RoboDK station: Group9-Robotics.rdk

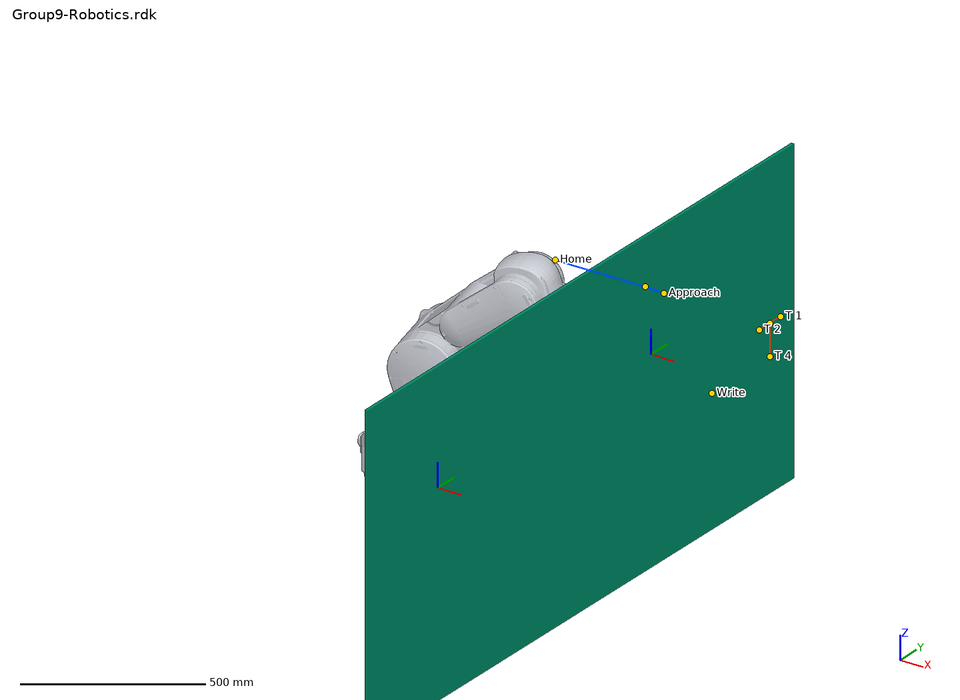
[picture v0: the station drawn from its stored meshes, robots at their saved joint values, targets as dots, program paths as lines]
Station ProjectWrite5 (saved by RoboDK 5.6.8). Poses are relative to the parent item; angles as X-Y-Z fixed-axis rotations.
Station parameters (name, value as stored): red, -1
  - frame Mitsubishi RV-7FR Base at (0, 0, 0) mm
    - robot Mitsubishi RV-7FR: 6 axes, payload 7 kg, reach 713 mm, repeatability 0.02 mm, weight 65 kg
        modified DH rows (alpha deg, a mm, theta deg, d mm): 0, 0, 0, 400; -90, 0, -90, 0; 0, 340, -90, 0; -90, 50, 0, 370; 90, 0, 0, 0; -90, 0, 180, 85
        joint limits [-240, -115, 0, -200, -120, -360] to [240, 125, 156, 200, 120, 360]; home [0, 0, 90, 0, 0, 0]; saved at [13.788, 47.313, 119.158, 14.166, -76.867, 176.718]
      - tool Tool, TCP at (0, 0, 283) mm, rotated rx 0 ry 0 rz -90 deg, size 100 x 89.2 x 281.5 mm
  - frame Frame 2 at (0, 1000, 0) mm
    - target Approach (Cartesian target) at (742, -1000, 790) mm, rotated rx 90 ry 0 rz 90 deg; joints [0, 0.675, 89.322, 180, -0.004, 0] of Mitsubishi RV-7FR
    - target Home (Cartesian target) at (386.81, -1000, 790) mm, rotated rx 90 ry 0 rz 90 deg; joints [0, -58.255, 121.519, 180, -26.736, 0] of Mitsubishi RV-7FR
    - target Write (Cartesian target) at (742, -775, 400) mm, rotated rx 90 ry 0 rz 90 deg; joints [31.031, 34.171, 112.413, 35.782, -61.843, 161.216] of Mitsubishi RV-7FR
    - target Retract (Cartesian target) at (680.67, -1000, 792.94) mm, rotated rx 90 ry 0 rz 90 deg; joints [0, -9.518, 98.336, 180, -1.182, 0] of Mitsubishi RV-7FR
    - target T 1 (Cartesian target) at (740, -450, 500) mm, rotated rx 0 ry 90 rz 0 deg; joints [55.927, 60.719, 47.204, 78.242, -57.788, -68.671] of Mitsubishi RV-7FR
    - target T 2 (Cartesian target) at (740, -550, 500) mm, rotated rx 0 ry 90 rz 0 deg; joints [50.421, 44.575, 75.507, 67.493, -56.542, -53.073] of Mitsubishi RV-7FR
    - target T 3 (Cartesian target) at (740, -500, 500) mm, rotated rx 0 ry 90 rz 0 deg; joints [53.351, 51.664, 63.311, 72.561, -57.241, -59.863] of Mitsubishi RV-7FR
    - target T 4 (Cartesian target) at (740, -500, 400) mm, rotated rx 0 ry 90 rz 0 deg; joints [53.351, 59.352, 66.003, 66.708, -60.867, -48.513] of Mitsubishi RV-7FR
  - object Board2mX1m at (740, -400, 1000) mm, rotated rx -90 ry 0 rz -90 deg, size 2000 x 1000 x 10 mm, geometry from Board2mX1m.STEP
  - program Prog1 (8 instructions, listed below)
  - Python program WriteRobodk (listed below)
  - program Prog3 (7 instructions, listed below)
  - Python program TimesNewRoman (listed below)
  - program Main Prog (3 instructions, listed below)
  - Python program WeldOff (listed below)
  - Python program WeldOn (listed below)
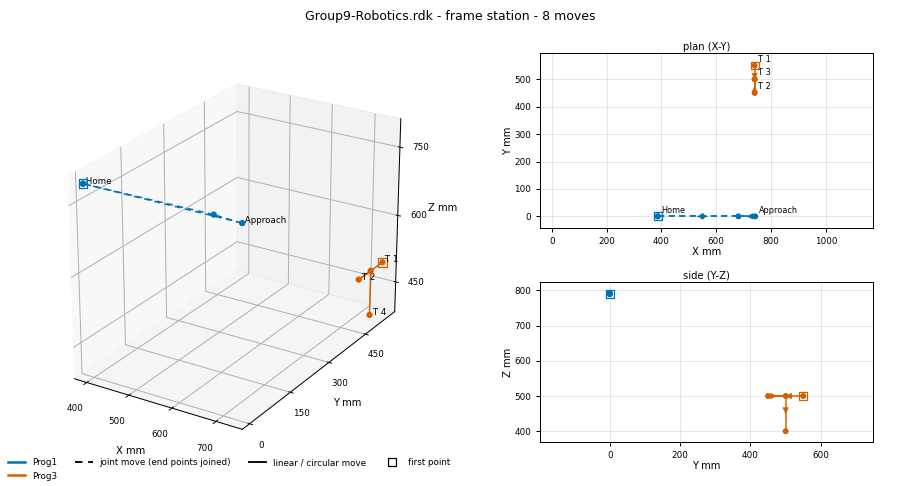
[picture p0: tool path of Group9-Robotics.rdk in frame station, 8 of 8 moves have a stored position in this frame; points joined in program order, loops and branches not executed]

--- program Prog1 (robot Mitsubishi RV-7FR) ---
  Set Ref.: Frame 2
  Set Tool: Tool
  MoveJ (Home)
  Call WeldOn(ON, ,red)
  MoveJ (Approach)
  MoveJ (Retract)
  MoveJ (Home)
  Call WeldOff

--- Python program WriteRobodk ---
# Type help("robodk.robolink") or help("robodk.robomath") for more information
# Press F5 to run the script
# Documentation: https://robodk.com/doc/en/RoboDK-API.html
# Reference:     https://robodk.com/doc/en/PythonAPI/robodk.html
# Note: It is not required to keep a copy of this file, your Python script is saved with your RDK project

# You can also use the new version of the API:
from robodk import robolink    # RoboDK API
from robodk import robomath    # Robot toolbox
RDK = robolink.Robolink()

# Forward and backwards compatible use of the RoboDK API:
# Remove these 2 lines to follow python programming guidelines
from robodk import *      # RoboDK API
from robolink import *    # Robot toolbox

program_name = 'Prog1'

robot = RDK.Item(" ",ITEM_TYPE_ROBOT)
frame = RDK.Item('Frame 2')
target = RDK.Item('Approach')
robot.setFrame(frame)

print(Pose_2_TxyzRxyz(target.Pose()))
txyz = Pose_2_TxyzRxyz(target.Pose())
print(txyz[0],txyz[1],txyz[2])

x = txyz[0]
y = txyz[1]
z = txyz[2]


program_item = RDK.Item(program_name, ITEM_TYPE_PROGRAM)

# Check if the program item is valid
if program_item.Valid():
    # Run the program
    program_item.RunProgram()

    print(f"Executing program: {program_name}")
else:
    print(f"Program not found: {program_name}")

--- program Prog3 (robot Mitsubishi RV-7FR) ---
  Set Ref.: Frame 2
  Set Tool: Tool
  Call WeldOn(ON, ,red)
  MoveJ (T 1)
  MoveL (T 2)
  MoveL (T 3)
  MoveL (T 4)

--- Python program TimesNewRoman ---
#zarady,muiz,chong
from robolink import *  # RoboDK's API
from robodk import *    # Math toolbox for robots
import csv              # to import excel file

# Opening Excel Files
file = open(r"C:\Users\USER\OneDrive - International Islamic University Malaysia\Desktop\BMCT\Robodk\Project\AdyChongMuiz.csv")
csvreader = csv.reader(file)
header = next(csvreader)
print(header)
rows = []
for row in csvreader:
    rows.append(row)

# Converting the values into floats
rows = [list(map(float, sublist)) for sublist in rows]
print(rows) # for verification of the float type

# Start the RoboDK API
RDK = Robolink()

# Get the robot
robot = RDK.Item('Select a Robot', ITEM_TYPE_ROBOT)
#print(RDK.ItemList())

if robot.Valid():
    print("Invalid targets. Exiting...")
    quit()

# Get the refference target by name :
target = RDK.Item('Write')
home = RDK.Item('Home')
target_pose = target.Pose()
xyz_ref = [target_pose.Pos()]
print(xyz_ref) # For verification of float types

robot.MoveJ(home)
robot.MoveJ(target)

print("Number of rows:", len(rows))


# Start engraving
for i in range(2994):
    # Calculate the new position
    x = xyz_ref[0][0]
    y = xyz_ref[0][1]- (rows[i][0]/2)
    z = xyz_ref[0][2]- (rows[i][1]/2)
    target_pose.setPos([x,y,z])
    robot.MoveJ(target_pose)


# Trigger a program call at the end of the moment
robot.RunInstruction('Program_Done')
print("Done Execute...")

--- program Main Prog (robot Mitsubishi RV-7FR) ---
  Call WeldOn(ON, ,red)
  Call TimesNewRoman
  Call WeldOff(-1)

--- Python program WeldOff ---
# This macro allows simulating the material deposition of a weld gun
# By default, this macro will activate the trace once it is called.
# Run the macro ArcEnd to stop the trace.
#
# The macros WeldOn, ArcEnd and Arc, all behave the same way, the only difference is the default behavior
# This behavior simmulates Fanuc Arc Welding and triggers appropriate output when using the customized post processor.
# Select ESC to clear the trace manually.
#
# It is possible to call WeldOn(ON) to simulate turning the material deposition ON or WeldOn(OFF) to stop simulating the gun
# Calling WeldOn(RESET) clears all displayed data.
# The macro will output spray gun statistics
#
# Optional:
# This macro can manage multiple guns and multiple colors.
# As an example, you can call this macro the following way:
#
# AcrStart(State, ToolName, Color)
#     State: [ON/OFF/RESET]
#     TorchName: The name of the tool. For example: Tool 1
#     Color: A named color or a hex color in the format: '#AARRGGBB'
#             Important: for full color definition you should provide Alpha channel first
#
# Examples:
#     WeldOn(ON)                 # Turn on the trace using the default color
#     WeldOn(OFF)                # Turn off the tool trace
#     WeldOn(ON, Tool 1, yellow) # Turn on the trace for tool 1 in yellow
#     WeldOn(ON, Tool 2, blue) # Turn on the trace for tool 2 in blue
#     WeldOn(OFF, Torch1)        # Turn off trace for Torch 1
#     WeldOn(ON, Torch1, #889900FF) # Turn on the trace for torch 2 in a violet color
#     WeldOn(ON, ,red)         # Turn on the trace for a generic torch in red color
#
# --------------------------------------------------------------
# This script shows how to create "spray" object in RoboDK that allows simulating particle deposition by using:
# RDK.Spray_Add(tool, object, options_command, volume, geometry)
#    tool: tool item (TCP) to use
#    object: object to project the particles
#    options_command (optional): string to specify options.
#    volume (optional): Matrix of parameters defining the volume of the spray gun
#    geometry (optional): Matrix of vertices defining the triangles.
#
# More information here:
# https://robodk.com/doc/en/PythonAPI/robodk.html#robodk.robolink.Robolink.Spray_Add
# https://robodk.com/doc/en/RoboDK-API.html
#
# The scripts ArcStart, ArcEnd and WeldOn and SpindleOn behave in a similar way, the only difference is the default behavior
# This behavior simmulates Fanuc Arc Welding and triggers appropriate output when using the customized post processor.
# Select ESC to clear the trace manually.
#
# Example scripts that use Spray_Add:
#     SpindleOn / SpindleOff    -> Turn trace On/Off
#     ArcOn / ArcOff            -> Turn trace On/Off
#     SprayOn / SprayOff        -> Simulate a spray given a workspace volume (for painting)
#     WeldOn / WeldOff          -> Support for multiple weld guns
#
#----------------------------------------------------------

# Constant variables for the first parameter:
ACTION_RESET = -1  # Same as: RESET (clear all traces)
ACTION_OFF = 0  # Same as: OFF (turn on)
ACTION_ON = 1  # Same as: ON (turn off)

# Define the default Action (ACTION_OFF to deactivate, ACTION_ON to activate, ACTION_RESET to clear any spray gun/trace)
# Setting it to None will display a message
Action = ACTION_OFF

# Define the default color as a named color or as #AARRGGBB (Alpha, Red, Green Blue)
# COLOR = 'blue'
COLOR = '#CC3344FF'  # AARRGGBB

# Use a specific tool as a spray gun
Tool_Name = None  # Use the active tool
#Tool_Name = 'Torch1'

# Use a specific object to project particles:
Object_Name = None  # Use the first object in the active reference frame
#Object_Name = 'Part'

# --------------------------------------------------
# Program start:
from robodk.robolink import *  # API to communicate with RoboDK
from robodk.robodialogs import *

RDK = Robolink()

# quit if we are not in simulation mode
if RDK.RunMode() != RUNMODE_SIMULATE:
    quit()

# Check command input (parameters passed in the call). This is the same as if we were doing a command line call passing parameters.
import sys
if len(sys.argv) > 1:
    Action_str = sys.argv[1].strip().upper()
    if 'ON' in Action_str:
        Action = ACTION_ON
    elif 'OFF' in Action_str:
        Action = ACTION_OFF
    elif 'RESET' in Action_str:
        Action = ACTION_RESET
    else:
        Action = int(Action_str)

    if len(sys.argv) > 2:
        Tool_Name = sys.argv[2].strip()
        if Tool_Name == '':
            Tool_Name = None

        if len(sys.argv) > 3:
            COLOR = sys.argv[3].lower().strip()

# Display summary
print("Applying action: " + str(Action))
print("Using tool: " + str(Tool_Name))
print("Using color: " + COLOR)

# Get any previously added spray gun simulations and display statistics (spray on the part vs spray falling out of the part)
info, data = RDK.Spray_GetStats()
n_sprays = data.size(1)
spray_id = -1
if n_sprays > 0 and Tool_Name is not None:
    spray_id = RDK.getParam(Tool_Name)
    if spray_id is None or Action == ACTION_ON or type(spray_id) == str or spray_id >= n_sprays:
        spray_id = -1

    print("Spray gun statistics:")
    print(info)
    print(data.tr())
    # # Diplay statistics
    # RDK.ShowMessage("Material used: %.1f%%<br>Material waisted: %.1f%%<br>Total particles: %.1f" % (data[1,0],data[2,0],data[3,0]), True)
    # # Clear previous spray
    # RDK.Spray_Clear()

# If the default Action is None, display a message to activate/deactivate the spray gun
if Action is None:
    print('Note: This macro can be called as ArcStart(1) or ArcStart(0) or ArcStart(-1)')
    entry = mbox('Turn gun ON or OFF', ('On', '1'), ('Off', '0'))
    if not entry:
        quit()
    Action = int(entry)

# Apply the desired action
if Action == ACTION_OFF:
    # Turn the gun off
    RDK.Spray_SetState(SPRAY_OFF, spray_id)

elif Action == ACTION_RESET:
    # Clear all spray simulations (same as pressing ESC key)
    RDK.Spray_Clear(spray_id)

elif Action == ACTION_ON:
    # Create a new spray gun object in RoboDK
    # by using RDK.Spray_Add(tool, object, options_command, volume, geometry)
    # tool: tool item (TCP) to use
    # object: object to project the particles
    # options_command (optional): string to specify options. Example:
    #     STEP=AxB: Defines the grid to be projected 1x1 means only one line of particle projection (for example, for welding)
    #     PARTICLE: Defines the shape and size of particle (sphere or particle), unless a specific geometry is provided:
    #       a- SPHERE(radius, facets)
    #       b- SPHERE(radius, facets, scalex, scaley, scalez)
    #       b- CUBE(sizex, sizey, sizez)
    #     RAND=factor: Defines a random factor factor 0 means that the particles are not deposited randomly
    #     ELLYPSE: defines the volume as an ellypse (default)
    #     RECTANGLE: defines the volume as a rectangle
    #     PROJECT: project the particles to the surface (default) (for welding, painting or scanning)
    #     NO_PROJECT: does not project the particles to the surface (for example, for 3D printing)
    #
    # volume (optional): Matrix of parameters defining the volume of the spray gun
    # geometry (optional): Matrix of vertices defining the triangles.

    if spray_id < 0:
        tool = 0  # auto detect active tool
        obj = 0  # auto detect object in active reference frame
        if Tool_Name is not None:
            tool = RDK.Item(Tool_Name, ITEM_TYPE_TOOL)

        if Object_Name is not None:
            obj = RDK.Item(Object_Name, ITEM_TYPE_OBJECT)
        # We can specify a given tool object and/or object
        #robot = RDK.Item("ABB IRB 2600-12/1.85", ITEM_TYPE_ROBOT)
        #tools = robot.Childs()
        #if len(tools) > 0:
        #    tool = tools[0]
        #obj = RDK.Item('object', ITEM_TYPE_OBJECT)

        # Create volume parameters
        options_command = "NO_PROJECT PARTICLE=SPHERE(2,8,1,1,1) STEP=1x0 RAND=0 COLOR=" + COLOR

        spray_id = RDK.Spray_Add(tool, obj, options_command)

    # Remember the ID of the spray gun for later
    if Tool_Name is not None:
        RDK.setParam(Tool_Name, spray_id)

    # Apply the state to activate the trace
    RDK.Spray_SetState(SPRAY_ON, spray_id)

--- Python program WeldOn ---
# This macro allows simulating the material deposition of a weld gun
# By default, this macro will activate the trace once it is called.
# Run the macro ArcEnd to stop the trace.
#
# The macros ArcStart, ArcEnd and WeldOn, SpindleOn, all behave in a similar way, the only difference is the default behavior
# This behavior simmulates Fanuc Arc Welding and triggers appropriate output when using the customized post processor.
# Select ESC to clear the trace manually.
#
# It is possible to call WeldOn(ON) to simulate turning the material deposition ON or WeldOn(OFF) to stop simulating the gun
# Calling WeldOn(RESET) clears all displayed data.
# The macro will output spray gun statistics
#
# Optional:
#     This macro can manage multiple guns and multiple colors.
#     As an example, you can call this macro the following way:
#
# WeldOn(State, ToolName, Color)
#     State: [ON/OFF/RESET]
#     TorchName: The name of the tool. For example: Tool 1
#     Color: A named color or a hex color in the format: '#AARRGGBB'
#             Important: for full color definition you should provide Alpha channel first
#
# Examples:
#     WeldOn(ON)                 # Turn on the trace using the default color
#     WeldOn(OFF)                # Turn off the tool trace
#     WeldOn(ON, Tool 1, yellow) # Turn on the trace for tool 1 in yellow
#     WeldOn(ON, Tool 2, blue) # Turn on the trace for tool 2 in blue
#     WeldOn(OFF, Torch1)        # Turn off trace for Torch 1
#     WeldOn(ON, Torch1, #889900FF) # Turn on the trace for torch 2 in a violet color
#     WeldOn(ON, ,red)         # Turn on the trace for a generic torch in red color
#
# --------------------------------------------------------------
# This script shows how to create "spray" object in RoboDK that allows simulating particle deposition by using:
# RDK.Spray_Add(tool, object, options_command, volume, geometry)
#    tool: tool item (TCP) to use
#    object: object to project the particles
#    options_command (optional): string to specify options.
#    volume (optional): Matrix of parameters defining the volume of the spray gun
#    geometry (optional): Matrix of vertices defining the triangles.
#
# More information here:
# https://robodk.com/doc/en/PythonAPI/robodk.html#robodk.robolink.Robolink.Spray_Add
# https://robodk.com/doc/en/RoboDK-API.html
#
# The scripts ArcStart, ArcEnd and WeldOn and SpindleOn behave in a similar way, the only difference is the default behavior
# This behavior simmulates Fanuc Arc Welding and triggers appropriate output when using the customized post processor.
# Select ESC to clear the trace manually.
#
# Example scripts that use Spray_Add:
#     SpindleOn / SpindleOff    -> Turn trace On/Off
#     ArcOn / ArcOff            -> Turn trace On/Off
#     SprayOn / SprayOff        -> Simulate a spray given a workspace volume (for painting)
#     WeldOn / WeldOff          -> Support for multiple weld guns
#
#----------------------------------------------------------

# Constant variables for the first parameter:
ACTION_RESET = -1  # Same as: RESET (clear all traces)
ACTION_OFF = 0  # Same as: OFF (turn on)
ACTION_ON = 1  # Same as: ON (turn off)

# Define the default Action (ACTION_OFF to deactivate, ACTION_ON to activate, ACTION_RESET to clear any spray gun/trace)
# Setting it to None will display a message
Action = ACTION_ON

# Define the default color as a named color or as #AARRGGBB (Alpha, Red, Green Blue)
# COLOR = 'blue'
COLOR = '#CC3344FF'  # AARRGGBB

# Use a specific tool as a spray gun
Tool_Name = None  # Use the active tool
#Tool_Name = 'Torch1'

# Use a specific object to project particles:
Object_Name = None  # Use the first object in the active reference frame
#Object_Name = 'Part'

# --------------------------------------------------
# Program start:
from robodk.robolink import *  # API to communicate with RoboDK
from robodk.robodialogs import *

RDK = Robolink()

# quit if we are not in simulation mode
if RDK.RunMode() != RUNMODE_SIMULATE:
    quit()

# Check command input (parameters passed in the call). This is the same as if we were doing a command line call passing parameters.
import sys
if len(sys.argv) > 1:
    Action_str = sys.argv[1].strip().upper()
    if 'ON' in Action_str:
        Action = ACTION_ON
    elif 'OFF' in Action_str:
        Action = ACTION_OFF
    elif 'RESET' in Action_str:
        Action = ACTION_RESET
    else:
        Action = int(Action_str)

    if len(sys.argv) > 2:
        Tool_Name = sys.argv[2].strip()
        if Tool_Name == '':
            Tool_Name = None

        if len(sys.argv) > 3:
            COLOR = sys.argv[3].lower().strip()

# Display summary
print("Applying action: " + str(Action))
print("Using tool: " + str(Tool_Name))
print("Using color: " + COLOR)

# Get any previously added spray gun simulations and display statistics (spray on the part vs spray falling out of the part)
info, data = RDK.Spray_GetStats()
n_sprays = data.size(1)
spray_id = -1
if n_sprays > 0 and Tool_Name is not None:
    spray_id = RDK.getParam(Tool_Name)
    if spray_id is None or Action == ACTION_ON or type(spray_id) == str or spray_id >= n_sprays:
        spray_id = -1

    print("Spray gun statistics:")
    print(info)
    print(data.tr())
    # # Diplay statistics
    # RDK.ShowMessage("Material used: %.1f%%<br>Material waisted: %.1f%%<br>Total particles: %.1f" % (data[1,0],data[2,0],data[3,0]), True)
    # # Clear previous spray
    # RDK.Spray_Clear()

# If the default Action is None, display a message to activate/deactivate the spray gun
if Action is None:
    print('Note: This macro can be called as ArcStart(1) or ArcStart(0) or ArcStart(-1)')
    entry = mbox('Turn gun ON or OFF', ('On', '1'), ('Off', '0'))
    if not entry:
        quit()
    Action = int(entry)

# Apply the desired action
if Action == ACTION_OFF:
    # Turn the gun off
    RDK.Spray_SetState(SPRAY_OFF, spray_id)

elif Action == ACTION_OFF:
    # Clear all spray simulations (same as pressing ESC key)
    RDK.Spray_Clear(spray_id)

elif Action == ACTION_ON:
    # Create a new spray gun object in RoboDK
    # by using RDK.Spray_Add(tool, object, options_command, volume, geometry)
    # tool: tool item (TCP) to use
    # object: object to project the particles
    # options_command (optional): string to specify options. Example:
    #     STEP=AxB: Defines the grid to be projected 1x1 means only one line of particle projection (for example, for welding)
    #     PARTICLE: Defines the shape and size of particle (sphere or particle), unless a specific geometry is provided:
    #       a- SPHERE(radius, facets)
    #       b- SPHERE(radius, facets, scalex, scaley, scalez)
    #       b- CUBE(sizex, sizey, sizez)
    #     RAND=factor: Defines a random factor factor 0 means that the particles are not deposited randomly
    #     ELLYPSE: defines the volume as an ellypse (default)
    #     RECTANGLE: defines the volume as a rectangle
    #     PROJECT: project the particles to the surface (default) (for welding, painting or scanning)
    #     NO_PROJECT: does not project the particles to the surface (for example, for 3D printing)
    #
    # volume (optional): Matrix of parameters defining the volume of the spray gun
    # geometry (optional): Matrix of vertices defining the triangles.

    if spray_id < 0:
        tool = 0  # auto detect active tool
        obj = 0  # auto detect object in active reference frame
        if Tool_Name is not None:
            tool = RDK.Item(Tool_Name, ITEM_TYPE_TOOL)

        if Object_Name is not None:
            obj = RDK.Item(Object_Name, ITEM_TYPE_OBJECT)
        # We can specify a given tool object and/or object
        #robot = RDK.Item("ABB IRB 2600-12/1.85", ITEM_TYPE_ROBOT)
        #tools = robot.Childs()
        #if len(tools) > 0:
        #    tool = tools[0]
        #obj = RDK.Item('object', ITEM_TYPE_OBJECT)

        # Create volume parameters
        options_command = "NO_PROJECT PARTICLE=SPHERE(2,8,1,1,1) STEP=1x0 RAND=0 COLOR=" + COLOR

        spray_id = RDK.Spray_Add(tool, obj, options_command)

    # Remember the ID of the spray gun for later
    if Tool_Name is not None:
        RDK.setParam(Tool_Name, spray_id)

    # Apply the state to activate the trace
    RDK.Spray_SetState(SPRAY_ON, spray_id)
